(* IEC 61131-3 sources: programs/VI-54/VI-54_20171205/VI-54_20171205/Stations/Screen/LseClass170718/Class/OrClass, 1 file *)

(* ---- OrClass.st ---- *)
(*!
<Class
	Name               = "OrClass"
	Revision           = "0.0"
	RealtimeTask       = "false"
	CyclicTask         = "false"
	BackgroundTask     = "false"
	Sigmatek           = "false"
	OSInterface        = "false"
	HighPriority       = "false"
	Automatic          = "false"
	UpdateMode         = "Prescan"
	SharedCommandTable = "true"
	Objectsize         = "(390,360)">
	<Channels>
		<Server Name="InvInputs" Visualized="true" Initialize="true" WriteProtected="false" Retentive="File"/>
		<Server Name="Result" Visualized="false" Initialize="false" WriteProtected="true" Retentive="false"/>
		<Client Name="Inp1" Required="true" Internal="false"/>
		<Client Name="Inp2" Required="true" Internal="false"/>
		<Client Name="Inp3" Required="true" Internal="false"/>
		<Client Name="Inp4" Required="true" Internal="false"/>
		<Client Name="Inp5" Required="true" Internal="false"/>
		<Client Name="Inp6" Required="true" Internal="false"/>
	</Channels>
</Class>
*)
OrClass : CLASS
  //Servers:
	Result 	: SvrChCmd_DINT;
	InvInputs 	: SvrCh_DINT;
  //Clients:
	Inp1 	: CltCh_DINT;
	Inp2 	: CltCh_DINT;
	Inp3 	: CltCh_DINT;
	Inp4 	: CltCh_DINT;
	Inp5 	: CltCh_DINT;
	Inp6 	: CltCh_DINT;
  //Variables:
  //Functions:

	FUNCTION VIRTUAL GLOBAL Result::Read
		VAR_OUTPUT
			output (EAX) 	: DINT;
		END_VAR;
  //Tables:
	FUNCTION @STD
		VAR_OUTPUT
			ret_code	: CONFSTATES;
		END_VAR;
	FUNCTION GLOBAL TAB @CT_;
END_CLASS;

FUNCTION VIRTUAL GLOBAL OrClass::Result::Read
	VAR_OUTPUT
		output (EAX) 	: DINT;
	END_VAR

  if IsClientConnected(#Inp1) then
    if InvInputs = 1 then
      Inp1 := (Inp1.Read() = 0);
    else
      Inp1 := Inp1.Read();
    end_if;
  end_if;
  if IsClientConnected(#Inp2) then
    if InvInputs = 1 then
      Inp2 := (Inp2.Read() = 0);
    else
      Inp2 := Inp2.Read();
    end_if;
  end_if;
  if IsClientConnected(#Inp3) then
    if InvInputs = 1 then
      Inp3 := (Inp3.Read() = 0);
    else
      Inp3 := Inp3.Read();
    end_if;
  end_if;
  if IsClientConnected(#Inp4) then
    if InvInputs = 1 then
      Inp4 := (Inp4.Read() = 0);
    else
      Inp4 := Inp4.Read();
    end_if;
  end_if;
  if IsClientConnected(#Inp5) then
    if InvInputs = 1 then
      Inp5 := (Inp5.Read() = 0);
    else
      Inp5 := Inp5.Read();
    end_if;
  end_if;
  if IsClientConnected(#Inp6) then
    if InvInputs = 1 then
      Inp6 := (Inp6.Read() = 0);
    else
      Inp6 := Inp6.Read();
    end_if;
  end_if;

  Result := (Inp1 | Inp2 | Inp3 | Inp4 | Inp5 | Inp6);

	output := Result;

END_FUNCTION
